// TIA Portal V20 export
DATA_BLOCK "DQ1"   // DB289
// stored: MemoryReserve 100
   VAR
      "EQUIPMENT LED LAMP RELAY ON" : Bool;
      SPARE1 : Bool;
      SPARE2 : Bool;
      "CLASS2 SMPS ALARM RESET" : Bool;
      SPARE3 : Bool;
      SPARE4 : Bool;
      SPARE5 : Bool;
      SPARE6 : Bool;
      SPARE7 : Bool;
      SPARE8 : Bool;
      SPARE9 : Bool;
      SPARE10 : Bool;
      SPARE11 : Bool;
      SPARE12 : Bool;
      SPARE13 : Bool;
      SPARE14 : Bool;
      SPARE15 : Bool;
      SPARE16 : Bool;
      SPARE17 : Bool;
      SPARE18 : Bool;
      SPARE19 : Bool;
      SPARE20 : Bool;
      SPARE21 : Bool;
      SPARE22 : Bool;
      SPARE23 : Bool;
      SPARE24 : Bool;
      SPARE25 : Bool;
      SPARE26 : Bool;
      SPARE27 : Bool;
      SPARE28 : Bool;
      SPARE29 : Bool;
      SPARE30 : Bool;
   END_VAR
BEGIN
END_DATA_BLOCK
